(* CODESYS project Tanque Industrial TON e TOF.project

Project tree, tasks and I/O mapping:
  Device : CODESYS Control Win V3, 3S - Smart Software Solutions GmbH, order no. 305021, version 3.5.11.30
    application Application
      libraries: Standard, * (System)
      task MainTask (cyclic, interval t#20ms, priority 1) calls PLC_PRG
      program PLC_PRG [LD]
      Symbols
*)

// Device/Application/PLC_PRG
PROGRAM PLC_PRG
VAR
	Encher:BOOL;
	Descarga:BOOL;
	Enchendo:BOOL;
	Esvaziando:BOOL;
	Valvula_Encher:BOOL;
	Valvula_Descarga:BOOL;
	Tempo_Encher:INT;
	Tempo_Esvaziar:INT; 
		
	TOF_0: TOF;
	tempo1: TIME;
	TON_0: TON;
	tempo2: TIME;
END_VAR

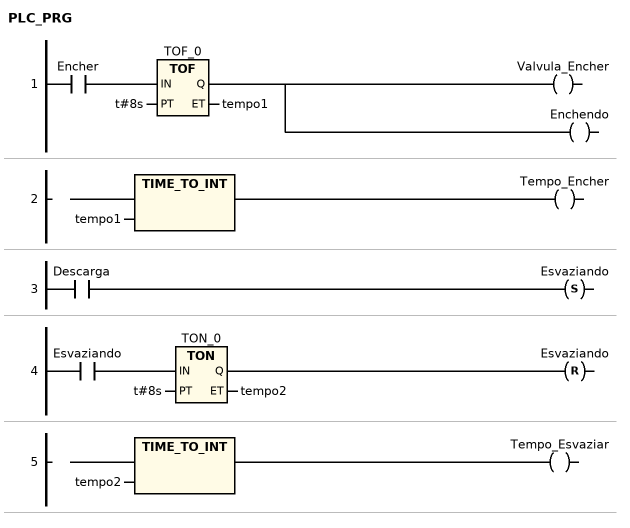
// NETWORK 1
TOF_0(IN := Encher, PT := t#8s, ET => tempo1); // TOF
Valvula_Encher := TOF_0.Q;
Enchendo := TOF_0.Q;

// NETWORK 2
Tempo_Encher := TIME_TO_INT(tempo1);

// NETWORK 3
Esvaziando S= Descarga;

// NETWORK 4
TON_0(IN := Esvaziando, PT := t#8s, ET => tempo2); // TON
Esvaziando R= TON_0.Q;

// NETWORK 5
Tempo_Esvaziar := TIME_TO_INT(tempo2);

END_PROGRAM
